// TIA Portal V20 export
DATA_BLOCK "DB_Alarm"   // DB14
// stored: Access Published, MemoryReserve 100, Namespace LineB1
   VAR
      "word" : Struct
         Line : Struct
            B1 : Struct
               Conveyor : Array[_.minB1.._.maxB1] of Word;
            END_STRUCT;
         END_STRUCT;
      END_STRUCT;
   END_VAR
BEGIN
END_DATA_BLOCK
